INTERFACE I_NciChannel_FeedTable EXTENDS I_NciChannelBase

PROPERTY IsChannelDone : BOOL
GET
END_GET
END_PROPERTY

PROPERTY IsFeedingDone : BOOL
GET
END_GET
END_PROPERTY

METHOD StartFeedTable
VAR_IN_OUT
    stTable : ST_NciFeedGroupTable;
END_VAR
END_METHOD

END_INTERFACE

(* stored: Version 1.1.0.1, ProductVersion 3.1.4024.15
   Itf I_NciChannel_FeedTable: Id {bdf92831-2e75-4c35-a24c-4989ea99c8c4}
   Property IsChannelDone: Id {4ead269f-09ad-4df7-8f7f-00024060bb5a}
   Get Get: Id {13cf23f8-6eeb-4112-a6fb-3a44675097ea}
   Property IsFeedingDone: Id {1ecd186c-8ec0-4aba-b014-9bd66a0385e4}
   Get Get: Id {f380b1a1-b2ef-4290-b619-22396bb326ad}
   Method StartFeedTable: Id {8ce29da5-6094-4383-a319-46ff66acdd31} *)
